{attribute 'pack_mode' := '4'}
TYPE ST_Filter_Current_Hexapod_Robot_InitData :
STRUCT
	Header: TComInitDataHdr;
	CallByHdr: TComInitDataElmHdr;
	CallBy: TctModuleCallByType;
	ExecutionSequenceHdr: TComInitDataElmHdr;
	ExecutionSequence: TctModuleExecutionSequenceType;
	StepSizeHdr: TComInitDataElmHdr;
	StepSize: TctStepSizeType;
	ExecuteModelCodeHdr: TComInitDataElmHdr;
	ExecuteModelCode: BOOL;
	ModelParametersHdr: TComInitDataElmHdr;
	ModelParameters: P_Filter_Current_Hexapod_Robo_T;
	ContextInfoArr_0_TaskOidHdr: TComInitDataElmHdr;
	ContextInfoArr_0_TaskOid: OTCID;
	ContextInfoArr_0_TaskPriorityHdr: TComInitDataElmHdr;
	ContextInfoArr_0_TaskPriority: UDINT;
	ContextInfoArr_0_TaskCycleTimeNsHdr: TComInitDataElmHdr;
	ContextInfoArr_0_TaskCycleTimeNs: UDINT;
	ContextInfoArr_0_TaskPortHdr: TComInitDataElmHdr;
	ContextInfoArr_0_TaskPort: UINT;
	ContextInfoArr_0_TaskSortOrderHdr: TComInitDataElmHdr;
	ContextInfoArr_0_TaskSortOrder: UDINT;
END_STRUCT
END_TYPE

(* stored: Version 1.1.0.1, ProductVersion 3.1.4020.12
   DUT ST_Filter_Current_Hexapod_Robot_InitData: Id {cb6c6a90-bde9-4b54-9668-7c8e75be2daf} *)
